FUNCTION_BLOCK CM_SensorAnalog
VAR_INPUT
	
	PI_ManualMode : BOOL;
	PI_AutoMode : BOOL;
	
	//ALARMS:
	PI_AlarmHighEnable : BOOL;
	PI_AlarmLowEnable : BOOL;
	PI_AlarmHighHighEnable : BOOL;
	PI_AlarmLowLowEnable : BOOL;
	PI_AlarmHighLimit : REAL;
	PI_AlarmLowLimit : REAL;
	PI_AlarmHighHighLimit : REAL;
	PI_AlarmLowLowLimit : REAL;
	
	PI_AlarmDelay_HH : INT;
	PI_AlarmDelay_H : INT;
	PI_AlarmDelay_L : INT;
	PI_AlarmDelay_LL : INT;
	
	PI_Alarmslatched : BOOL;
	PI_AlarmsAknowlegded : BOOL;
	
	PI_PV :DINT;
	PI_PV_REAL : REAL;
	PI_PV_MANUAL : REAL;
	
	ENABLE_SCALING : BOOL;
	PI_PV_MAX_IN : INT;
	PI_PV_MIN_IN : INT;
	PI_PV_MAX_OUT : INT;
	PI_PV_MIN_OUT : INT;
END_VAR
VAR_OUTPUT
	
	PO_PV_SCALED : REAL;
	PO_PV_REAL : REAL;

	
	PO_ALARM_HH : BOOL;
	PO_ALARM_H : BOOL;
	PO_ALARM_L : BOOL;
	PO_ALARM_LL : BOOL;
	
	
END_VAR
VAR
	scale : Tc2_ControllerToolbox.FB_CTRL_SCALE;
	scaleParams : ST_CTRL_SCALE_PARAMS;
	
	prg_scan_HH : INT; // used for alarm delay
	prg_scan_H : INT; // used for alarm delay
	prg_scan_L : INT; // used for alarm delay
	prg_scan_LL : INT; // used for alarm delay
	
	Alarm_Ack_HH : BOOL;
	Alarm_Ack_H : BOOL;
	Alarm_Ack_L : BOOL;
	Alarm_Ack_LL : BOOL;
	
END_VAR
VAR_IN_OUT
	CM_UDT_CTRL : Udt_CM_SensorAnalog;
	Plant_control : Udt_PlantControl;
END_VAR

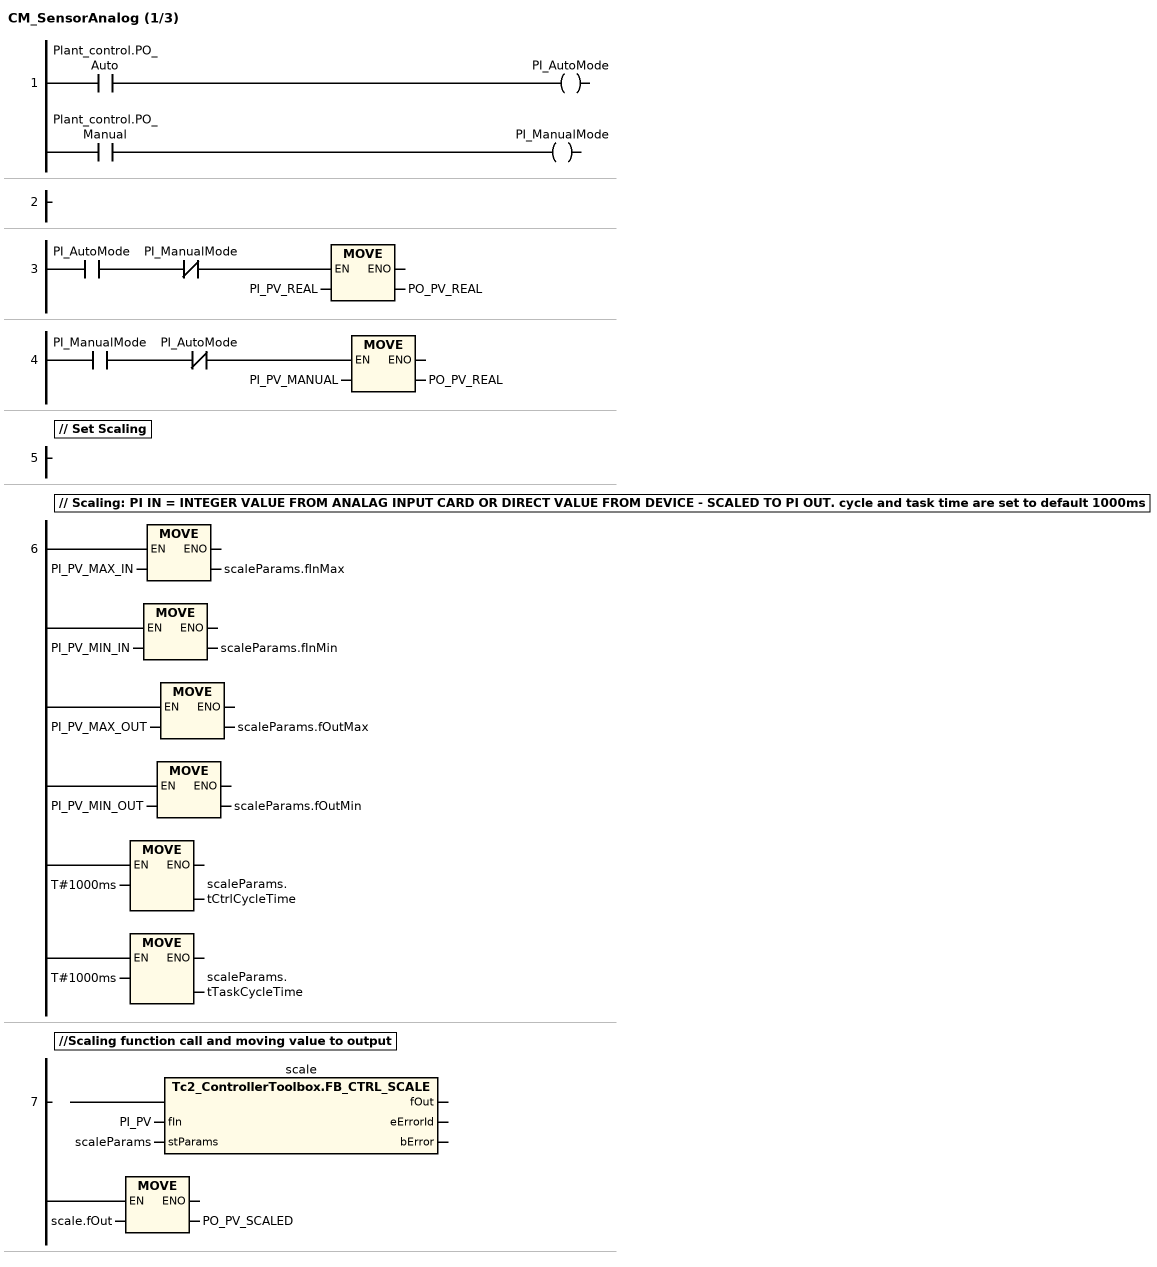
// NETWORK 1
PI_AutoMode := Plant_control.PO_Auto;
PI_ManualMode := Plant_control.PO_Manual;

// NETWORK 2

// NETWORK 3
IF PI_AutoMode AND NOT PI_ManualMode THEN PO_PV_REAL := PI_PV_REAL; END_IF

// NETWORK 4
IF PI_ManualMode AND NOT PI_AutoMode THEN PO_PV_REAL := PI_PV_MANUAL; END_IF

// NETWORK 5
// label: // Set Scaling

// NETWORK 6
// label: // Scaling: PI IN = INTEGER VALUE FROM ANALAG INPUT CARD OR DIRECT VALUE FROM DEVICE - SCALED TO PI OUT. cycle and task time are set to default 1000ms
scaleParams.fInMax := PI_PV_MAX_IN;
scaleParams.fInMin := PI_PV_MIN_IN;
scaleParams.fOutMax := PI_PV_MAX_OUT;
scaleParams.fOutMin := PI_PV_MIN_OUT;
scaleParams.tCtrlCycleTime := T#1000ms;
scaleParams.tTaskCycleTime := T#1000ms;

// NETWORK 7
// label: //Scaling function call and moving value to output
scale(fIn := PI_PV, stParams := scaleParams); // Tc2_ControllerToolbox.FB_CTRL_SCALE
PO_PV_SCALED := scale.fOut;

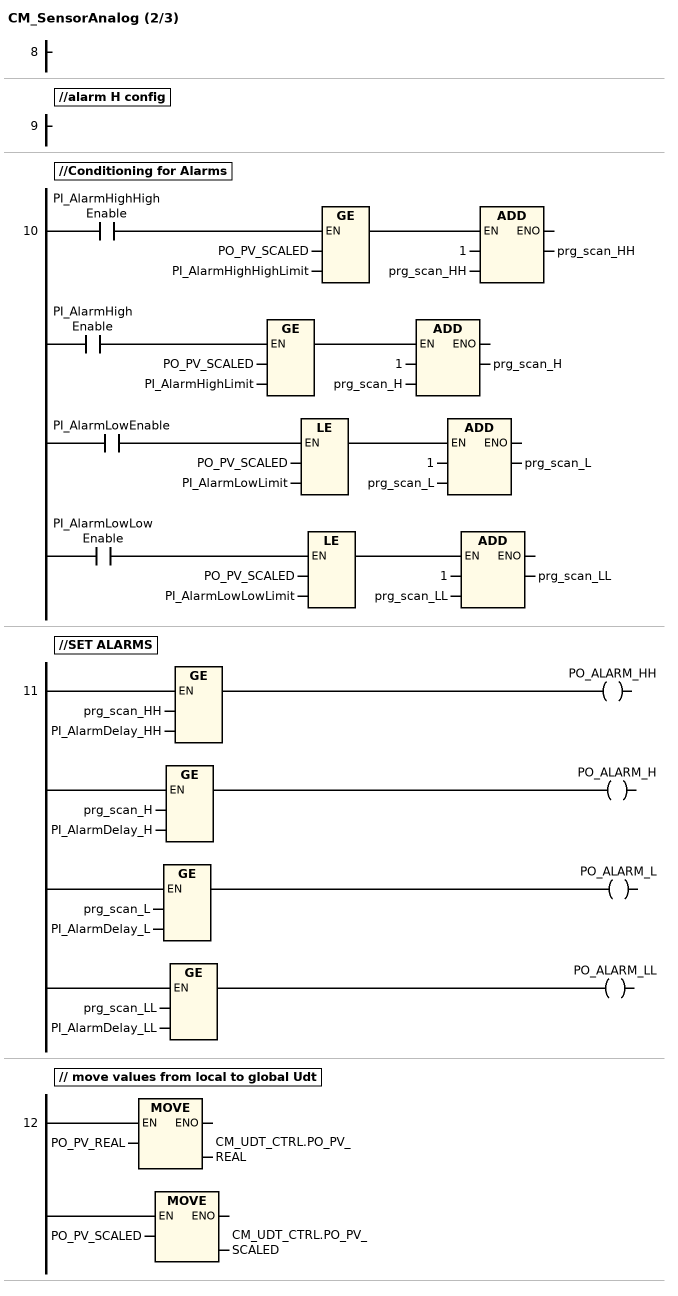
// NETWORK 8

// NETWORK 9
// label: //alarm H config

// NETWORK 10
// label: //Conditioning for Alarms
IF PI_AlarmHighHighEnable AND PO_PV_SCALED >= PI_AlarmHighHighLimit THEN prg_scan_HH := 1 + prg_scan_HH; END_IF
IF PI_AlarmHighEnable AND PO_PV_SCALED >= PI_AlarmHighLimit THEN prg_scan_H := 1 + prg_scan_H; END_IF
IF PI_AlarmLowEnable AND PO_PV_SCALED <= PI_AlarmLowLimit THEN prg_scan_L := 1 + prg_scan_L; END_IF
IF PI_AlarmLowLowEnable AND PO_PV_SCALED <= PI_AlarmLowLowLimit THEN prg_scan_LL := 1 + prg_scan_LL; END_IF

// NETWORK 11
// label: //SET ALARMS
PO_ALARM_HH := prg_scan_HH >= PI_AlarmDelay_HH;
PO_ALARM_H := prg_scan_H >= PI_AlarmDelay_H;
PO_ALARM_L := prg_scan_L >= PI_AlarmDelay_L;
PO_ALARM_LL := prg_scan_LL >= PI_AlarmDelay_LL;

// NETWORK 12
// label: // move values from local to global Udt
CM_UDT_CTRL.PO_PV_REAL := PO_PV_REAL;
CM_UDT_CTRL.PO_PV_SCALED := PO_PV_SCALED;

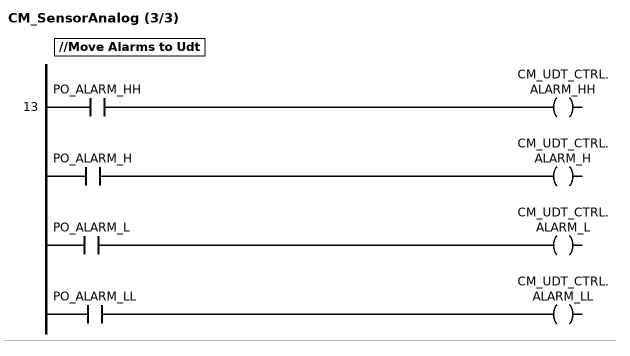
// NETWORK 13
// label: //Move Alarms to Udt
CM_UDT_CTRL.ALARM_HH := PO_ALARM_HH;
CM_UDT_CTRL.ALARM_H := PO_ALARM_H;
CM_UDT_CTRL.ALARM_L := PO_ALARM_L;
CM_UDT_CTRL.ALARM_LL := PO_ALARM_LL;

END_FUNCTION_BLOCK

(* stored: Version 1.1.0.1, ProductVersion 3.1.4024.13
   POU CM_SensorAnalog: Id {91247847-bd09-4fb6-8a55-10da55afbf65}, SpecialFunc None *)
